// Mitsubishi GX Works2 project: a7   PLC: Q02/Q02H

PROGRAM MAIN
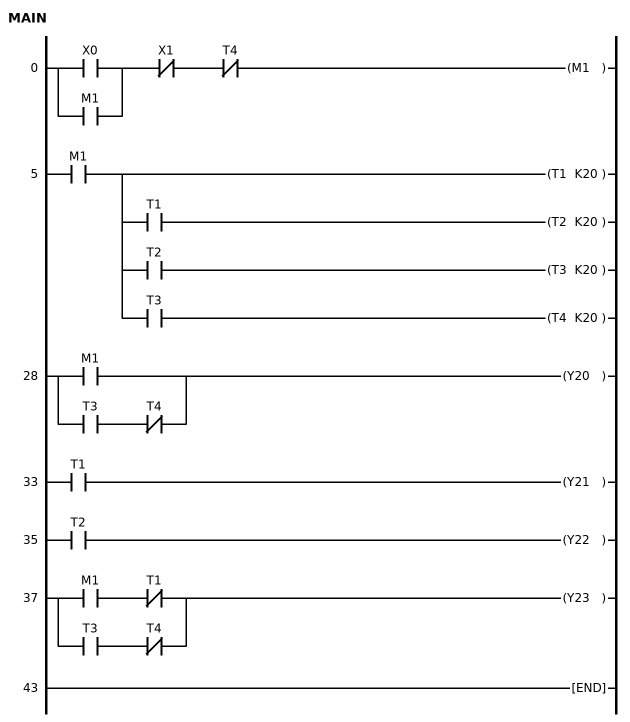
0     LD      X0
      OR      M1
      ANI     X1
      ANI     T4
      OUT     M1
5     LD      M1
      OUT     T1 K20
      MPS
      AND     T1
      OUT     T2 K20
      MRD
      AND     T2
      OUT     T3 K20
      MPP
      AND     T3
      OUT     T4 K20
28    LD      M1
      LD      T3
      ANI     T4
      ORB
      OUT     Y20
33    LD      T1
      OUT     Y21
35    LD      T2
      OUT     Y22
37    LD      M1
      ANI     T1
      LD      T3
      ANI     T4
      ORB
      OUT     Y23
43    END
END_PROGRAM
